FUNCTION_BLOCK ThreeConCtl (* Composite Function Block Type *)
  (* Standard: 61499-2 *)
  (* Version 0.2, 2003-12-05, JHC, Rockwell Automation, Renamed from NEWCOMPFB. *)
  (* Version 0.1, 2002-01-08, JHC, Rockwell Automation, Added DLY FB as example. *)
  (* Version 0.0, 2000-05-27, JHC, Rockwell Automation *)
  (* Compiler header: package fb.rt.cs725; *)
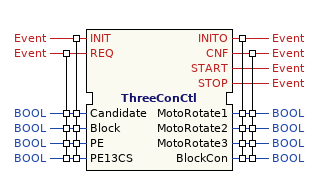
  EVENT_INPUT
    INIT WITH Candidate, Block, PE, PE13CS; (* Initialization Request *)
    REQ WITH Block, Candidate, PE, PE13CS; (* Normal Execution Request *)
  END_EVENT
  EVENT_OUTPUT
    INITO WITH MotoRotate1, MotoRotate2, MotoRotate3, BlockCon; (* Initialization Confirm *)
    CNF WITH MotoRotate1, MotoRotate2, MotoRotate3, BlockCon; (* Execution Confirmation *)
    START;
    STOP;
  END_EVENT
  VAR_INPUT
    Candidate : BOOL;
    Block : BOOL;
    PE : BOOL;
    PE13CS : BOOL;
  END_VAR
  VAR_OUTPUT
    MotoRotate1 : BOOL;
    MotoRotate2 : BOOL;
    MotoRotate3 : BOOL;
    BlockCon : BOOL;
  END_VAR
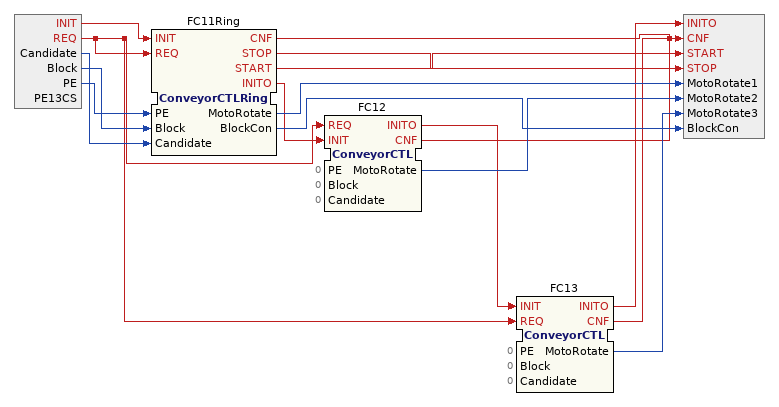
  FBS
    FC12 : ConveyorCTL(PE := 0, Block := 0, Candidate := 0);
    FC13 : ConveyorCTL(PE := 0, Block := 0, Candidate := 0);
    FC11Ring : ConveyorCTLRing;
  END_FBS
  EVENT_CONNECTIONS
    FC12.INITO TO FC13.INIT;
    FC13.INITO TO INITO;
    FC13.CNF TO CNF;
    REQ TO FC12.REQ;
    REQ TO FC13.REQ;
    FC12.CNF TO CNF;
    INIT TO FC11Ring.INIT;
    REQ TO FC11Ring.REQ;
    FC11Ring.CNF TO CNF;
    FC11Ring.STOP TO STOP;
    FC11Ring.START TO START;
    FC11Ring.INITO TO FC12.INIT;
  END_CONNECTIONS
  DATA_CONNECTIONS
    FC13.MotoRotate TO MotoRotate3;
    FC12.MotoRotate TO MotoRotate2;
    PE TO FC11Ring.PE;
    Block TO FC11Ring.Block;
    Candidate TO FC11Ring.Candidate;
    FC11Ring.MotoRotate TO MotoRotate1;
    FC11Ring.BlockCon TO BlockCon;
  END_CONNECTIONS
END_FUNCTION_BLOCK
